# B&R Automation Studio project Lab_1
Automation Studio 4.5.2.102

## Configuration Config1

CPU 4PP065.0571-P74, AutomationRuntime D4.52, Build 4.1.2, Vc V4.52.0

### Task classes (Cpu.sw)
```
Cyclic#1:
  Program <- Program.prg
Binaries: udbdef, TCData, ashwd, User, asfw, arconfig, sysconf, Role, ashwac, iomap
Libraries: Library
```

### Hardware
```
4PP065_0571_P74 : 4PP065.0571-P74 v1.2.0.0
  Connector IF5:
    ActivateDevice = 1
  ConfigurationID = Pract1_Config1
  Simulation = 1
```

## Logical view

### Library Logical/Libraries/Library (ANSIC)

#### Library.fun - Exported functions and function blocks
```iecst
FUNCTION_BLOCK FB_Integrator
	VAR_INPUT
		in : {REDUND_UNREPLICABLE} REAL;
	END_VAR
	VAR_OUTPUT
		out : REAL;
	END_VAR
	VAR
		dt : REAL;
	END_VAR
END_FUNCTION_BLOCK

FUNCTION_BLOCK FB_Regulator
	VAR_INPUT
		e : REAL;
	END_VAR
	VAR_OUTPUT
		u : REAL;
	END_VAR
	VAR
		k_p : REAL;
		k_i : REAL;
		integrator : FB_Integrator;
		iyOLD : REAL;
		max_abs_value : REAL;
		dt : REAL;
	END_VAR
END_FUNCTION_BLOCK

FUNCTION_BLOCK FB_Motor
	VAR_INPUT
		u : REAL;
	END_VAR
	VAR_OUTPUT
		w : REAL;
		phi : REAL;
	END_VAR
	VAR
		integrator : FB_Integrator;
		Tm : REAL;
		ke : REAL;
		dt : REAL;
	END_VAR
END_FUNCTION_BLOCK
```

#### FB_Integrator.c
```c
#include <bur/plctypes.h>
#ifdef __cplusplus
	extern "C"
	{
#endif
	#include "Library.h"
#ifdef __cplusplus
	};
#endif
/* TODO: Add your comment here */
void FB_Integrator(struct FB_Integrator* inst)
{
	if (inst==0)
		return;
	inst->out += inst->in*inst->dt;
}
```

#### FB_Regulator.c
```c
#include <bur/plctypes.h>
#ifdef __cplusplus
	extern "C"
	{
#endif
	#include "Library.h"
#ifdef __cplusplus
	};
#endif
/* TODO: Add your comment here */
void FB_Regulator(struct FB_Regulator* inst)
{

	REAL up;
	REAL ui;
	REAL u_raw;
	REAL u_lim;

	if (inst->dt <= 0.0f) inst->dt = 0.01f;
	if (inst->max_abs_value <= 0.0f) inst->max_abs_value = 24.0f;

	up = inst->k_p * inst->e;

	if (up >  inst->max_abs_value) up =  inst->max_abs_value;
	if (up < -inst->max_abs_value) up = -inst->max_abs_value;

	inst->integrator.dt = 1.0f;
	inst->integrator.in = inst->k_i * inst->dt * inst->e + inst->iyOLD;
	FB_Integrator(&inst->integrator);
	ui = inst->integrator.out;

	u_raw = up + ui;

	u_lim = u_raw;
	if (u_lim >  inst->max_abs_value) u_lim =  inst->max_abs_value;
	if (u_lim < -inst->max_abs_value) u_lim = -inst->max_abs_value;

	inst->iyOLD = u_lim - u_raw;

	inst->u = u_lim;
}
```

#### FB_Motor.c
```c
#include <bur/plctypes.h>
#ifdef __cplusplus
	extern "C"
	{
#endif
	#include "Library.h"
#ifdef __cplusplus
	};
#endif
/* TODO: Add your comment here */
void FB_Motor(struct FB_Motor* inst)
{
	if (inst==0)
		return ;
	REAL u_norm = inst->u / inst->ke;
	REAL din = (u_norm - inst->integrator.out) / inst->Tm;

	inst->integrator.in = din;
	FB_Integrator(&inst->integrator);
	inst->w = inst->integrator.out;

	inst->phi += inst->w * inst->dt;
}
```

### Program Logical/Program

#### Variables.var
```iecst
VAR
	Tzh : REAL;
	fb_motor : FB_Motor;
	fb_regulator : FB_Regulator;
	Enable : BOOL;
	Speed : REAL;
	fb_motor_2 : FB_Motor;
	Counter : USINT;
END_VAR
```

#### Cyclic.c
```c
#include <bur/plctypes.h>
#include <Library.h>

#ifdef _DEFAULT_INCLUDES
	#include <AsDefault.h>
#endif

void _CYCLIC ProgramCyclic(void)
{
	Counter ++;
	if (Counter > 100)
	{
		Speed = 90.0;
		Enable = 1;
	}
	if (Counter > 250)
	{
		Speed = 0.0;
	}
	fb_motor_2.u = Enable ? (Speed * fb_motor_2.ke) : 0.0;
	FB_Motor(&fb_motor_2);

	if (Enable)
	{
		fb_regulator.e = Speed - fb_motor.w;
		FB_Regulator(&fb_regulator);

		fb_motor.u = fb_regulator.u;
		FB_Motor(&fb_motor);
	}
	else
	{
		fb_motor.u = 0.0;
		FB_Motor(&fb_motor);
	}
}
```

#### Init.c
```c
#include <bur/plctypes.h>

#ifdef _DEFAULT_INCLUDES
	#include <AsDefault.h>
#endif

void _INIT ProgramInit(void)
{
	fb_motor.Tm = 0.05;
	fb_motor.ke = 0.05;
	fb_motor.integrator.dt = 0.01;
	fb_motor.integrator.out = 0.0;
	fb_motor.phi = 0.0;

	fb_motor_2.Tm = 0.05;
	fb_motor_2.ke = 0.05;
	fb_motor_2.integrator.dt = 0.01;
	fb_motor_2.integrator.out = 0.0;
	fb_motor_2.phi = 0.0;

   Tzh = 0.02;

	fb_regulator.k_p = fb_motor.ke * fb_motor.Tm / Tzh;
	fb_regulator.k_i = fb_motor.ke / Tzh;
	fb_regulator.max_abs_value = 24.0;
	fb_regulator.max_abs_value = 24.0;
	fb_regulator.integrator.dt = 0.01;
	fb_regulator.integrator.out = 0.0;

	Counter = 0;
	Speed = 0;
	Enable = 0;

}
```

Listed in the project but not available here: Logical/Libraries/Library/Types.typ, Logical/Libraries/Library/Constants.var
